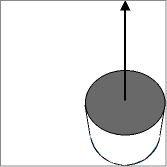
VISUALIZATION VISU_Tube_Top_3  // 167x167
VAR_IN_OUT
	azi : LREAL;
END_VAR
    Ellipse (90,100 70x65)
        p2858320360: azi
    Polygon (85,100) (165,100) (162,126) (160,135) (156,145) (151,152) (144,159) (134,163) (124,165) (111,162) (101,155) (95,147) (90,135)
        p2858320360: azi
    Ellipse (85,70 80x65)
        p2858320360: azi
    Polygon (120,10) (125,0) (130,10)
        p2858320360: azi
    Polyline (125,100) (125,10)
        p2858320360: azi
    Polyline (160,135) (165,105)
        p2858320360: azi
    Polyline (90,135) (85,105)
        p2858320360: azi
END_VISUALIZATION

(* stored: Version 1.1.0.1, ProductVersion 3.1.4018.5
   Visu VISU_Tube_Top_3: Id {dd1e61ed-a5c3-4f4b-b90a-80170171516c} *)
